PROGRAM FiveRung
VAR
	FromSqLogic: BOOL;
	Trigger: BOOL;
	Safe: BOOL;
	TimeoutFail: BOOL;
	EStopOK: BOOL;
	AutoMode: BOOL;
	InPosition: BOOL;
	ManualMode: BOOL;
	Pushbutton: BOOL;
	Command: BOOL;
	Sensor: BOOL;
	FaultTimer: BOOL;
	TON_FaultTimer: TON;
	TimeoutFault: BOOL;
	FaultReset: BOOL;
END_VAR

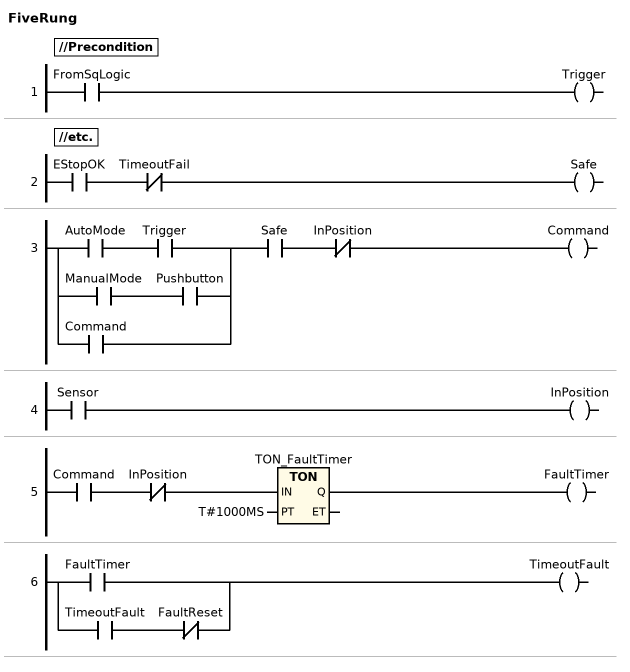
// NETWORK 1
// label: //Precondition
Trigger := FromSqLogic;

// NETWORK 2
// label: //etc.
Safe := EStopOK AND NOT TimeoutFail;

// NETWORK 3
Command := (AutoMode AND Trigger OR ManualMode AND Pushbutton OR Command) AND Safe AND NOT InPosition;

// NETWORK 4
InPosition := Sensor;

// NETWORK 5
TON_FaultTimer(IN := Command AND NOT InPosition, PT := T#1000MS); // TON
FaultTimer := TON_FaultTimer.Q;

// NETWORK 6
TimeoutFault := FaultTimer OR TimeoutFault AND NOT FaultReset;

END_PROGRAM

(* stored: Version 1.1.0.1, ProductVersion 3.1.4024.10
   POU FiveRung: Id {22d443e9-f0ed-4b62-9008-6991d3b6918a}, SpecialFunc None *)
